// TIA Portal project "Aufgabe_2_002_mCopilot" (V20)
// *** This TIA Portal project underwent AI modifications via the Siemens Engineering Copilot. ***

(* hardware
DEVICE "S7-1200 G2 station_1"  S7-1200 G2 Station
   slot 0: "Rack_0"  S71200G2 Rack  Rack  V1.0
   slot 1: "PLC_1"  CPU 1212C DC/DC/DC  6ES7 212-1AG50-0XB0  V1.0
*)

// ===== PLC "PLC_1"  CPU 1212C DC/DC/DC =====

VAR_GLOBAL   // PLC tag table "Default tag table"
   "S1" AT %I0.0 : Bool;
   "S2" AT %I0.1 : Bool;
   "S3" AT %I0.2 : Bool;
   "S4" AT %I0.3 : Bool;
   "M1" AT %Q0.0 : Bool;
   "M2" AT %Q0.1 : Bool;
   "M3" AT %Q0.2 : Bool;
   "M4" AT %Q0.3 : Bool;
   "Clock_Byte" AT %MB0 : Byte;
   "Clock_10Hz" AT %M0.0 : Bool;
   "Clock_5Hz" AT %M0.1 : Bool;
   "Clock_2.5Hz" AT %M0.2 : Bool;
   "Clock_2Hz" AT %M0.3 : Bool;
   "Clock_1.25Hz" AT %M0.4 : Bool;
   "Clock_1Hz" AT %M0.5 : Bool;
   "Clock_0.625Hz" AT %M0.6 : Bool;
   "Clock_0.5Hz" AT %M0.7 : Bool;
   "VarOverflow" AT %Q0.4 : Bool;
END_VAR

VAR_GLOBAL CONSTANT   // PLC tag table "Default tag table"
   "WARNING_THRESHOLD" : Int := 100;
END_VAR

// folder: Instances

DATA_BLOCK "InstBaggageAmountMonitoring"   // DB3
{ S7_Optimized_Access := 'TRUE' }
VERSION : 0.1
// stored: InstanceOfName FB_BaggagesCounting
"FB_BaggagesCounting"
BEGIN
END_DATA_BLOCK

// folder: (top level)

FUNCTION_BLOCK "FB_BaggagesCounting"   // FB22, SCL
{ S7_Optimized_Access := 'TRUE' }
VERSION : 0.1
   VAR_INPUT
      baggageDetect : Bool;   // Sensor S4
   END_VAR
   VAR_OUTPUT
      amountOfBaggage : USInt;   // Current counting value
      lineFull : Bool;   // LineFull Flag
   END_VAR
   VAR
      statAmount : UInt;
      statLineFull : Bool;
      statBaggageDetection : Bool;
   END_VAR
BEGIN
   REGION BLOCK INFO HEADER
       //===============================================================================
       //-------------------------------------------------------------------------------
       // Title:            FB_CountingBaggages
       // Comment/Function: This Block is counting the baggages when baggage detect sensor is triggered.
       // Library/Family:   N.A
       // Author:           ---
       // Tested with:      S7-1200 G2/CPU 1212C DC/DC/DC FW 1.0 
       // Engineering:      TIA Portal V20
       // Requirements:     --- 
       //-------------------------------------------------------------------------------
       // Change log table:
       // Version  | Date       | Expert in charge        | Changes applied
       //----------|------------|-------------------------|-----------------------------
       // 01.00.00 | 15.12.2025 |          N.N            | First released version
       //===============================================================================
   END_REGION BLOCK INFO HEADER

   REGION DESCRIPTION  
       (/*Purpose:
   This FB is used for roughly counting baggage on circular conveyor belt when the sensor is triggered. 
   A line full flag will be output when the count reaches the threshold and current count will be reset.
   This flag is used to remind operators of the full status.

   Usage:
   - Input 'baggageDetect' is used for counting the passed baggage number.
   - The 'lineFull' output will set to TRUE after the amount of baggage is larger than 300.
   - The 'amountOfBaggage' output is set by internal variable 'statAmount'.*/)

   END_REGION DESCRIPTION

   REGION INPUT
       #statBaggageDetection := #baggageDetect;
   END_REGION INPUT



   REGION PROCESSING
       // Detect whether the sensor for baggage detection is triggered. Then increase the amount by 1.
       IF #statBaggageDetection THEN
           #statAmount := #statAmount + 1;
       END_IF;

       // When the amount is larger than 300, the lineFull flag will be set to TRUE.
       IF #statAmount > 300 THEN
           #lineFull := TRUE;  
           #statAmount := 0;
       END_IF;
   END_REGION PROCESSING

   REGION OUTPUT 
       //Transfer internal value into output
       #amountOfBaggage := #statAmount;
       #lineFull := #statLineFull;
   END_REGION
END_FUNCTION_BLOCK

FUNCTION "FC_Check" : Void   // FC1, SCL
{ S7_Optimized_Access := 'TRUE' }
VERSION : 0.1
BEGIN
   //Funktionsinhalt nur zur Ueberpruefung der korrekten Verknuepfung des Projekts,
   //mit dem Engineering Copilot
   //
   //Rechenaufgabe
   //Berechne das Produkt von 9 und 4
END_FUNCTION

ORGANIZATION_BLOCK "Main"   // OB1, LAD, ProgramCycle
TITLE = "Main Program Sweep (Cycle)"
{ S7_Optimized_Access := 'TRUE' }
VERSION : 0.1
   VAR_INPUT
      Initial_Call : Bool;   // Initial call of this OB
      Remanence : Bool;   // =True, if remanent data are available
   END_VAR
BEGIN

REGION Network 1: FB_BaggagesCounting
   // Zaehlung des Gepaecks auf dem Ringfoerderband. Die Gepaeckerkennung mit Sensor S4 wird mittels eines periodischen Signals, mit einer Frequenz von 1 Hz, simuliert.
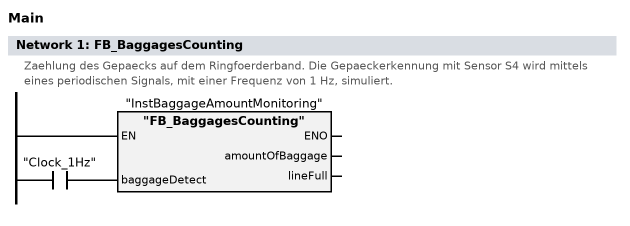
   RUNG wire#powerrail
      "InstBaggageAmountMonitoring"(baggageDetect := wire#w1, amountOfBaggage =>, lineFull =>)
   END_RUNG
   RUNG wire#powerrail
      Contact( "Clock_1Hz" )
   END_RUNG wire#w1
   // the same network as SCL:
   "InstBaggageAmountMonitoring"(baggageDetect := "Clock_1Hz");   // "FB_BaggagesCounting"
END_REGION
END_ORGANIZATION_BLOCK

// ===== library types =====

// folder: LGF/7 Signal generators

FUNCTION_BLOCK "LGF_Frequency"   // FB10024, SCL
TITLE = LGF_Frequency
{ S7_Optimized_Access := 'TRUE' }
AUTHOR : Siemens_Industry_Support
FAMILY : LGF
NAME : LGF_Frequency
// This function generates a signal that changes between the values `FALSE` and `TRUE` depending on a defined frequency and a pulse pause ratio. / Diese Funktion generiert ein Signal, das in Abhängigkeit von einer definierten Frequenz und einem Pulspausenverhältnis, zwischen den Werten `FALSE` und `TRUE` wechselt.
   VAR_INPUT
      frequency : Real := 0.0;   // Clock frequency in Hz. / Taktfrequenz in Hz.
      pulsePauseRatio : Real := 1.0;   // Pulse pause ratio (standard: 1.0 corresponds to 1:1). / Pulspausenverhältnis (Standard: 1.0 entspricht 1:1).
   END_VAR
   VAR_OUTPUT
      clock : Bool;   // Output changes with defined frequency. / Ausgang wechselt mit definierter Frequenz.
      countdown : Time;   // Remaining time of the current `clock` state. / Verbleibende Zeit des aktuellen Zustands von `clock`.
   END_VAR
   VAR
      instTofTimePulse : TOF_TIME;   // Timer instance for the Pulse signal (Period of time the clock signal is true)
      instTofTimePause : TOF_TIME;   // Timer instance for the Pause signal (Period of time the clock signal is false)
      statFrequencyOld : Real;   // Static Old/Current value of the frequency input
      statPulsePauseRatioOld : Real;   // Static Old/Current value of the pulsePauseRatio input
      statTimePulse : Time;   // Static calculated for me the pulse duration of the clock
      statTimePause : Time;   // Static calculated for me the pause duration of the clock
   END_VAR
   VAR_TEMP
      tempPulseRate : Real;   // Static calculation of pulse rate - needed for passing value between calculations
      tempPauseRate : Real;   // Static calculation of pause rate - needed for passing value between calculations
      tempCountdown : Time;   // Static countdown until next ON/OFF value of the clock signal
   END_VAR
   VAR CONSTANT
      ZERO : Real := 0.0;   // Numeric zero constant
      ZERO_TIME : Time := T#0ms;   // Time zero constant
      SECOND_IN_MS : Real := 1000.0;   // One second written in miliseconds. Needed in calculation in formulas
      ONE : Real := 1.0;   // 100% - One hundred procent / 100% - Einhundert Prozent
   END_VAR
BEGIN
   REGION Block info header
     //=============================================================================
     // SIEMENS AG / (c)Copyright 2017
     //-----------------------------------------------------------------------------
     // Title:            LGF_Frequency
     // Comment/Function: This function generates a signal that changes between the values `FALSE` and `TRUE` depending on a defined frequency and a pulse pause ratio.
     // Library/Family:   LGF(Library General Functions)
     // Author:           Siemens Digital Industry Support
     // Tested with:      S7-PLCSIM Advanced V2.0 SP1
     // Engineering:      TIA Portal V15 Update 2
     // Restrictions:     ENO disabled - error handling done by error and status
     // Requirements:     PLC (S7-1200 / S7-1500)
     //-------------------------------------------------------------------------------
     // Change log table:
     // Version  | Date       | Expert in charge       | Changes applied
     //----------|------------|------------------------|------------------------------
     // 01.00.00 19.08.2015  Siemens Industry Online Support
     //                      First released version
     // 01.01.00 25.05.2016  Siemens Industry Online Support
     //                      New function: pulse pause ratio
     // 01.01.01 26.05.2016  Siemens Industry Online Support
     //                      Add comments
     // 01.01.02 02.01.2017  Siemens Industry Online Support
     //                      Upgrade: TIA Portal V14 Update 1
     // 01.01.03 17.08.2018  Siemens Industry Online Support
     //                      Upgrade: TIA V15 Update 2
     // 01.01.04 23.11.2018  Siemens Industry Online Support
     //                      Upgrade: TIA V15.1
     // 01.00.07 20.09.2019  Simatic Systems Support
     //                      Code refactoring, regions and more comments added
     // 03.00.00 23.04.2020  Simatic Systems Support
     //                      Set version to V3.0.0, harmonize the version of the whole library
     // 03.00.01 15.02.2021  Simatic Systems Support
     //                      Insert documentation
     //=============================================================================
   END_REGION Block info header

   REGION DESCRIPTION
     (/*The `clock` output is a Boolean value that toggles at the desired frequency. The `pulsePauseRatio` input is used to set the pulse pause ratio.

   The output `countdown` outputs the remaining time of the current state of `clock`.

   If the desired frequency or pulse pause ratio is less than or equal to `0.0`, the output `clock` = FALSE and `countdown` = `0s`.

   ------

   #### Example

   ![LGF_Frequency](LGF_Frequency.png "LGF_Frequency")

   ---

   Note
   :    The `clock` of the FB LGF_Frequency depends on the cycle time of the OB
   Main. To increase the accuracy, the FB can also be called in a cyclic interrupt
   OB with a low time interval.
   Der Ausgang `clock` ist ein boolescher Wert, der in der gewünschten Frequenz toggelt. Über den Eingang `pulsePauseRatio` wird das Pulspausenverhältnis eingestellt.

   Der Ausgang `countdown` gibt die verbleibende Zeit des aktuellen Zustands von `clock` aus.

   Falls die gewünschte Frequenz oder das Pulspausenverhältnis kleiner oder gleich `0.0` ist, ist der Ausgang `clock` = FALSE und `countdown` = `0s`.

   ------

   #### Beispiel

   ![LGF_Frequency](LGF_Frequency.png "LGF_Frequency")

   ---

   Hinweis
   :    Der Takt (`clock`) des FB LGF_Frequency ist abhängig von der Zykluszeit des OB Main. Um die Genauigkeit zu erhöhen, kann der FB auch in einem Weckalarm-OB (Cyclic Interrupt OB) mit niedrigem Zeittakt aufgerufen werden.*/)
   END_REGION DESCRIPTION

   REGION Calculation of settings and program execution
     // If input <= 0.0 the block is disabled
     IF (#frequency <= #ZERO) OR (#pulsePauseRatio <= #ZERO) THEN
       #clock := FALSE;
       #tempCountdown := #ZERO_TIME;
     ELSE

       //Calculating function frequency and pulse pause ratio only when an input is changed
       IF #statFrequencyOld <> #frequency OR #statPulsePauseRatioOld <> #pulsePauseRatio THEN
         RESET_TIMER(TIMER := #instTofTimePause);
         RESET_TIMER(TIMER := #instTofTimePulse);

         #tempPulseRate := #pulsePauseRatio / (#pulsePauseRatio + #ONE); // Calculate pulse rate   
         #tempPauseRate := #ONE - #tempPulseRate;                      // Calculate pause rate   
         #statTimePulse := UDINT_TO_TIME(REAL_TO_UDINT((#SECOND_IN_MS * #tempPulseRate / #frequency))); // Calculate pulse time   
         #statTimePause := UDINT_TO_TIME(REAL_TO_UDINT((#SECOND_IN_MS * #tempPauseRate / #frequency))); // Calculate pause time
         #statFrequencyOld := #frequency;
         #statPulsePauseRatioOld := #pulsePauseRatio;
       END_IF;

       //Two time off-delay timers that are resetting each other on expiration
       #instTofTimePulse(IN := NOT #instTofTimePause.Q,
                         PT := #statTimePulse);

       //If timer for pulse is running, remaining time of the PULSE is calculated
       #tempCountdown := #statTimePulse - #instTofTimePulse.ET;

       #instTofTimePause(IN := #instTofTimePulse.Q,
                         PT := #statTimePause);

       //If timer for pulse is NOT running, remaining time of the PAUSE is calculated
       IF #tempCountdown = #ZERO_TIME THEN
         #tempCountdown := #statTimePause - #instTofTimePause.ET;
       END_IF;

     END_IF;
   END_REGION

   REGION Writing to outputs
     // Assigning value of the pulse timer to the clock output
     #clock := #instTofTimePulse.Q;
     #countdown := #tempCountdown;
     //ENO mechanism is not used - forced to true.
     ENO := TRUE;
   END_REGION
END_FUNCTION_BLOCK